{attribute addProperty BoxType "IODEVICETYPE_ETHERCATPROT"}
{attribute addProperty Id "boxesboxes_C34C4083340324254A_0076_AMP8000_0030_0103AMP8000_8C7527D258473SyncUnitsSyncUnits_3FA29F3C21627InputsInputs_C75D3FEC1280160OutputsOutputs_47D1E803848106InfoDataInfoData_45F98C5022428"}
{attribute addProperty CRC "2374790677"}
{attribute addProperty SizeInBites "37184"}
{attribute addProperty SizeInBytes "4648"}
TYPE EtherCAT_Master_Duplicates_8D8C6E15 :
STRUCT
	{attribute addProperty Name "boxes"}
	boxes : boxes_C34C4083;
	{attribute addProperty Name "A_0076_AMP8000_0030_0103"}
	A_0076_AMP8000_0030_0103 : AMP8000_8C7527D2;
	{attribute addProperty Name "SyncUnits"}
	SyncUnits : SyncUnits_3FA29F3C;
	{attribute addProperty Name "Inputs"}
	Inputs : Inputs_C75D3FEC;
	{attribute addProperty Name "Outputs"}
	Outputs : Outputs_47D1E803;
	{attribute addProperty Name "InfoData"}
	InfoData : InfoData_45F98C50;
END_STRUCT
END_TYPE

(* stored: Version 1.2.0.0, ProductVersion 3.1.4024.9
   DUT EtherCAT_Master_Duplicates_8D8C6E15: Id {8d403662-d02d-43d6-a68f-d75b723dbc64} *)
